// TIA Portal V20 export
TYPE "typeEm4Standard"
// stored: Access Published, Namespace Unit1
   STRUCT
      commands { ExternalWritable := 'False'} : "Unit1.typeEm4Commands";
      monitoring { ExternalWritable := 'False'} : "Unit1.typeEm4Monitoring";
   END_STRUCT;
END_TYPE
